FUNCTION_BLOCK FB_ExtractiveOutletControl
VAR_INPUT
	onOffValveCommand : BOOL;
	controlValveCommands : ST_ExtractiveControlValveCommands;
	controlValveParameters : ST_ExtractiveControlValveParameters;
END_VAR
VAR_OUTPUT
	onOffValveOpen : BOOL;
	onOffValveButtonCommand	: BOOL;
	controlValveClose	: BOOL;
	controlValveOpen	: BOOL;
	controlValveCurrentOpenPercentage : DINT;
	calibrateDone : BOOL;
END_VAR
VAR
	TON_OpenValve : TOF;
	TON_CloseValve : TOF;
	calibrate : BOOL;
	ControlValveStateMachine : FB_ControlValveStateMachine;
	onOffValveButton : FB_ValveTrigger;
END_VAR

//onOffValveOpen := onOffValveCommand;
onOffValveButton(
			openCommand := onOffValveCommand);
onOffValveButtonCommand := onOffValveButton.buttonCommand;
onOffValveOpen := onOffValveButton.isOpen;


ControlValveStateMachine(
						controlValveCommands := controlValveCommands,
						controlValveParameters := controlValveParameters,
						closeControlValve => controlValveClose,
						openControlValve => controlValveOpen,
						currentControlValveOpenPercentage => controlValveCurrentOpenPercentage,
						calibrateDone => calibrateDone);

END_FUNCTION_BLOCK

(* stored: Version 1.1.0.1, ProductVersion 3.1.4024.9
   POU FB_ExtractiveOutletControl: Id {c4646b40-ee7c-48e1-846d-cd0fb4b976bb}, SpecialFunc None *)
